Universal Robots PolyScope program: cottonMotorOn.urp

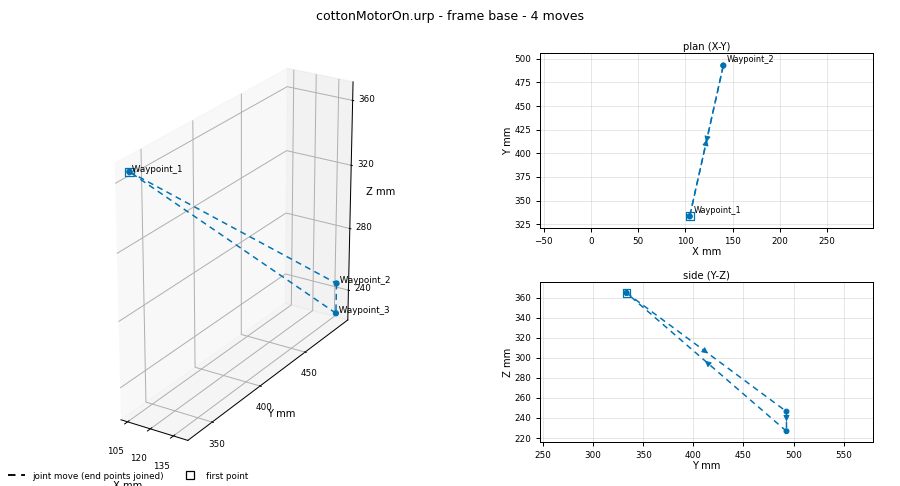
[picture p0: tool path of cottonMotorOn.urp in frame base, 4 of 6 moves have a stored position in this frame; points joined in program order, loops and branches not executed]
Program cottonMotorOn (installation=default directory=/programs/DavidMelin createdIn=5.12.4.1101661 lastSavedIn=5.12.4.1101661 robotSerialNumber=20225502378)
Calibrated DH parameters: a=[0.00022, -0.425328, -0.389701, 0.000059, 0.000065, 0]; d=[0.162608, 0.803456, 9.992211, -10.662202, 0.099702, 0.099559]; alpha=[1.570756, 0.001543, 0.004316, 1.570651, -1.570122, 0]; deltaTheta=[0, 0.002917, 0.116094, -0.119008, 0, -0.000001]
Robot Program (runOnlyOnce=true)
  MoveJ speed 60 deg/s, acceleration 80 deg/s^2 (useActiveTCP=true) feature=Base
    Waypoint Waypoint (Variable): variable=cotonHomePos
  URCap Gripper (Robotiq_Grippers, Robotiq Inc.) dataModel(position=100.0, force=0.0, speed=0.0, positionInDouble=100.0, forceInDouble=0.0, speedInDouble=0.0, slaveIds=[9], blocking=true)
  MoveJ speed 60 deg/s, acceleration 80 deg/s^2 (useActiveTCP=true) feature=Base
    Waypoint Waypoint_1: TCP in base x=104.65 y=333.28 z=364.789 mm, rx=-2.4906 ry=0.0958 rz=-0.1131 rad; joints [98.536, -64.728, -139.702, -29.678, 79.085, 9.451] deg
    Waypoint Waypoint_2: TCP in base x=140.283 y=492.919 z=246.408 mm, rx=-2.3951 ry=0.1183 rz=-0.0956 rad; joints [90.495, -106.57, -127.634, 6.507, 83.867, 3.943] deg
    Waypoint Waypoint_3: TCP in base x=140.261 y=492.93 z=226.81 mm, rx=-2.3949 ry=0.1183 rz=-0.0956 rad; joints [90.496, -109.342, -128.316, 9.967, 83.855, 3.946] deg
    Waypoint Waypoint_4: TCP in base x=104.681 y=333.271 z=364.78 mm, rx=-2.4906 ry=0.0959 rz=-0.1132 rad; joints [98.531, -64.728, -139.703, -29.68, 79.085, 9.451] deg
    Waypoint Waypoint (Variable): variable=cotonHomePos
